TYPE CyclicAxis_Error_typ :
	STRUCT
		ErrorID : UDINT ;
		ErrorText : STRING[2048];(*ARRAY[0..3]OF STRING[79]*) (*Error Text*)
		ErrorEntry: Eh_ErrorEntry_typ;
	END_STRUCT
END_TYPE

(* stored: Version 1.1.0.1, ProductVersion 3.1.4024.3
   DUT CyclicAxis_Error_typ: Id {4b7b3877-e2fc-0838-1024-7c0d110921c3} *)
